FUNCTION F_Temp_Write_Value : ST_Modbus_Send_Frame
VAR_INPUT
	Module_Number	:WORD;
	Command_Index	:WORD;
	Write_Value		:WORD;
END_VAR
VAR
END_VAR

F_Temp_Write_Value.StartAddress	:= Command_Index;
F_Temp_Write_Value.sendQuantity	:= 1;
F_Temp_Write_Value.SendData[0]	:= Write_Value;

END_FUNCTION

(* stored: Version 1.1.0.1
   POU F_Temp_Write_Value: Id {f8555c32-2600-4397-926c-cc4e887709e3}, SpecialFunc None *)
